// Return TRUE if the value is None.
// Optionally carries the value over to nOut for further processing.
FUNCTION IsNone : BOOL
VAR_INPUT
    nIn : Result; // Result variable to check for None
END_VAR
VAR_OUTPUT
    nOut : Result; // Carries the input value for further use
END_VAR

IsNone := nIn = 0;
nOut := nIn;

END_FUNCTION

(* stored: Version 1.1.0.1
   POU IsNone: Id {45d926e7-4340-49c1-9630-09ea933bc1ee}, SpecialFunc None *)
